{attribute 'qualified_only'}
VAR_GLOBAL
	gCanIf_TxMsg         AT %Q* : CAN_IFACE_QUEUE;
	gCanIf_RxMsg         AT %I* : CAN_IFACE_QUEUE;
END_VAR

(* stored: Version 1.1.0.1
   GVL EL6751_GVLs: Id {be69125a-6d33-4cc5-81a5-c4172fc8b04f} *)
